// TIA Portal V17 export
// export: Created 2025-03-05T07:59:43.6218373Z, ExportSetting WithDefaults, DisplayName Totally Integrated Automation Portal, DisplayVersion V17 Update 8, DisplayName TIA Portal Openness, DisplayVersion V17 Update 8, DisplayName TIA Portal Version Control Interface, DisplayVersion V17, DisplayName SINAMICS Startdrive Advanced, DisplayVersion V17 SP2, DisplayName SINAMICS Startdrive G110M, G120, G120C, G120D, G120P, G115D, DisplayVersion V17 SP2, DisplayName SINAMICS Startdrive G130, G150, S120, S150, SINAMICS MV, S210, DisplayVersion V17 SP2, DisplayName STEP 7 Professional, DisplayVersion V17 Update 8, DisplayName SINUMERIK ONE STEP 7 Toolbox, DisplayVersion V17 Update 12, DisplayName SINUMERIK 840D sl STEP 7 Toolbox, DisplayVersion V17 Update 12, DisplayName STEP 7 Safety, DisplayVersion V17 Update 6, DisplayName WinCC Advanced, DisplayVersion V17 Update 8
DATA_BLOCK "DB335_EXTENDED_M_CODE_UNIT_02_STA_2"   // DB335
{ DB_Accessible_From_OPC_UA := 'FALSE' }
AUTHOR : ETXETAR
FAMILY : MCODES
VERSION : 1.0
// stored: AutoNumber false, DBAccessibleFromOPCUA false, DBAccessibleFromWebserver true, InstanceOfName FB331_M_CODE_EXTENDED, InstanceOfType FB
"FB331_M_CODE_EXTENDED"
   // VAR_INPUT
   //    NC_Chan_Num_Chan : Int;
   // END_VAR
   // VAR RETAIN
   //    INDEX : Int;
   //    M_code : Array[100..999] of Bool;
   // END_VAR
BEGIN
END_DATA_BLOCK
